Staubli VAL3: oHeater.pgx

public program oHeater(num nState (dimensions=1), num nDuration (dimensions=1))
begin
  switch nState
    case 0
      dioSet(oHeater,0)
      if (taskStatus("heating")==1)
        taskKill("heating")
      endIf
    break
    case 1
      taskCreate "heating",3,oHeaterTask(nDuration)
    break
    default
    break
  endSwitch
end
